Fanuc KAREL source: ks00034.KL

-- PROVISIONAL review KL for V1013-1; original PC SHA256 492633dd69818497c119d819b4d4f34ffe46e0f77abde78f1f64e1311d705880
-- Incomplete behavior may be omitted. Consult companion uncertainty JSON. Do not deploy.
PROGRAM KS00034
%NOLOCKGROUP
VAR
  FLAG : BOOLEAN
  N : INTEGER
  STATUS : INTEGER
  PN : STRING[80]
  VN : STRING[80]
-- UNRESOLVED_DECL A type=00201c
-- UNRESOLVED_DECL B type=00201c
BEGIN
  -- UNRESOLVED_PC offsets 5-13; opcodes 3F,75
  -- UNRESOLVED_PC offsets 18-27; opcodes 3F,75
  -- UNRESOLVED_PC offsets 32-70; opcodes 27,22,22,2A,22,2A,22,22,AF
  -- UNRESOLVED_PC offsets 75-79; opcodes 7F
END KS00034
